FUNCTION_BLOCK Q_ChangeObjectLabel (* Command Change Object Label( Part 6 - F.50 ) *)
  (* Standard: ISO 11783-6; Description: Copyright (c) 2022 HR Agrartechnik GmbH This program and the accompanying materials are made available under the terms of the Eclipse Public License 2.0 which is available at https://www.eclipse.org/legal/epl-2.0/ SPDX-License-Identifier: EPL-2.0 see Description Tab *)
  (* Version 1.0, 2022-07-08, Franz Höpfinger, HR Agrartechnik GmbH *)
  PACKAGE isobus::UT::Q;
  IMPORT isobus::UT::Q::const::IDs::ID_NULL;
  (* Documentation:
  Command Change Object Label( Part 6 - F.50 )
   This command is used by a Working Set to change a label of an object.
   Valid values for u16ObjId (the object to label)
   The Change Object Label command (F.50) carries, in bytes 2,3, the Object ID of the object to associate a label with. Per Annex F.51 (response error Bit 0) and B.21, the addressed object must be listed in the Object Label Reference List object — i.e. any pool object (e.g. a Soft Key, WorkingSet or input object) whose ID is an entry of the Object Label Reference List.
   Implementation note (VTClientHelper): the C function iso_is_object_label_refer_list_id instead accepts only the ObjectLabelReferList type range (the Object Label Reference List object's own ID range). This is a known deviation from the Annex F.50 semantics — the FB commands only IDs in this range:
    - ObjectLabelReferList: 40000 – 40999
    ID_NULL (65535) is not a command target but can be used in INIT to deactivate the FB. Any ID outside this range is invalid for commanding.
   Activate / Deactivate
   The FB is deactivated by default. It becomes active when INIT provides a valid object label Object ID. Sending INIT with ID_NULL (65535) deactivates the FB again. This toggle can be repeated arbitrarily.
    - INIT + ID_NULL (65535): FB deactivated, STATUS="DEACTIVATED", s16result=VT_E_DEACTIVATED (-40)
   - INIT + valid object label ID: FB activated, STATUS="initialized", s16result=VT_E_NO_ERR (0). If a REQ was buffered before, it is executed immediately.
   - INIT + invalid ID: STATUS="ERROR: Invalid Object ID (not an object label object)", s16result=VT_E_INVALID_OBJECT_ID (-132)
    REQ Handling
    - REQ before any INIT: Buffered, STATUS="Buffered: INIT not yet completed", s16result=VT_E_NOT_READY (-131)
   - REQ while deactivated (INIT came with NULL or invalid ID): STATUS shows the actual deactivation reason, s16result=VT_E_DEACTIVATED (-40) or VT_E_INVALID_OBJECT_ID (-132)
   - REQ while active: Command sent to VT, result reflected in CNF
    param[in] {objectID, uint16_t}
   Object ID of object to associate label with. Use ID_NULL (65535) to deactivate the FB. Use a valid object label object ID to activate.
   param[in] {labelStringObjectID, uint16_t}
   Object ID of a String Variable object that contains the label string (32 characters maximum) or FFFF if no text is supplied
   param[in] {fontType, uint8_t}
   Font type (ignored if String Variable object reference is NULL or the string contains a WideString)
   param[in] {graphicalDesignatorObjectID, uint16_t}
   Object ID of an object to be used as a graphic representation of the object label or FFFF16 if no designator supplied.
   Return Values (s16result):
   int16_t
    - VT_E_NO_ERR (0) - OK
   - VT_E_DEACTIVATED (-40) - FB deactivated (INIT received with ID_NULL)
   - VT_E_INVALID_OBJECT_ID (-132) - Object ID is invalid (not an object label object)
   - VT_E_NOT_READY (-131) - Buffered: INIT not yet completed
   - VT_E_OVERFLOW (-6) - buffer overflow
   - VT_E_NOACT (-8) - Command not possible in current state
   - VT_E_NO_INSTANCE (-21) - No VT client available
   - VT_E_ISO_INSTANCE_INVALID (-129) - Identifier for instance (connection) invalid
   - VT_E_NOT_ALIVE (-130) - Identifier for instance valid, but VT Dead.
    Instanz-Eindeutigkeit (Instance Uniqueness)
   Dieser Baustein erfordert Instanz-Eindeutigkeit bezüglich u16ObjId. Es darf im gesamten Programm nur eine Instanz von Q_ChangeObjectLabel für dieselbe Ziel-Objekt-ID existieren. Eine zweite Instanz auf dieselbe Objekt-ID wird bei INIT deaktiviert (STATUS = "This objID is already in use").
  *)
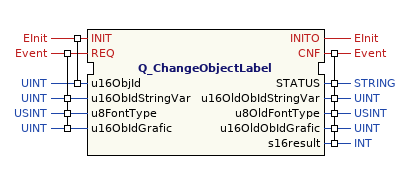
  EVENT_INPUT
    INIT : EInit WITH u16ObjId; (* Service Initialization *)
    REQ WITH u16ObIdStringVar, u8FontType, u16ObIdGrafic; (* Service Request *)
  END_EVENT
  EVENT_OUTPUT
    INITO : EInit; (* Initialization Confirm *)
    CNF WITH STATUS, u16OldObIdStringVar, u8OldFontType, u16OldObIdGrafic, s16result, u16OldObIdStringVar, u8OldFontType, u16OldObIdGrafic; (* Confirmation of Requested Service *)
  END_EVENT
  VAR_INPUT
    u16ObjId : UINT := ID_NULL; (* Object ID *)
    u16ObIdStringVar : UINT := ID_NULL; (* Object ID of a String Variable object that contains the label string (32 characters maximum) or FFFF if no text is supplied *)
    u8FontType : USINT; (* Font type (ignored if String Variable object reference is NULL or the string contains a WideString ) *)
    u16ObIdGrafic : UINT := ID_NULL; (* Object ID of an object to be used as a graphic representation of the object label or FFFF16 if no designator supplied *)
  END_VAR
  VAR_OUTPUT
    STATUS : STRING; (* Service Status *)
    u16OldObIdStringVar : UINT; (* Old Object ID of a String Variable object that contains the label string (32 characters maximum) or FFFF if no text is supplied *)
    u8OldFontType : USINT; (* Old value for attribute *)
    u16OldObIdGrafic : UINT;
    s16result : INT; (* retval see description *)
  END_VAR
END_FUNCTION_BLOCK
